// TIA Portal V18 export
FUNCTION "AHUTargetUnitStatesCtrl" : Void   // FC60104, LAD
{ S7_Optimized_Access := 'TRUE' }
VERSION : 0.1
// Operation Modes                                                 Unit State
// 0=Protection                                                         0=Stopped
// 1=Economy                                                           1=Checking-up  
// 2=PreComfort                                                       2=Preheating
// 3=Comfor                                                              3=Starting 
// 4=Auto(Scheduler)                                              4=RecirculatingOperation
//                                                                                 5=Economy Operation                                                                                                                                            6=PreComfort Operation 
//                                                                                 7=Comfort  operation
//                                                                                 8=Stopping
//                                                                                 9=Blocking
// stored: AutoNumber false, IsIECCheckEnabled false, SetENOAutomatically false, UDAEnableTagReadback false
   VAR_INPUT
      iUnitID : Int;
      cTargetOpMode : Byte;
      cActualOpMode : Byte;
      xStartRequest : Bool;
      xBlockRequest : Bool;
   END_VAR
   VAR_OUTPUT
      cTargetUnitState : Byte;
   END_VAR
BEGIN

REGION Network 1 (SCL)
   CASE #cActualOpMode OF
       0:                                                  // OpMode is OFF(Protection)
           IF #xBlockRequest THEN                               // Stop by alarm      
               #cTargetUnitState := 9;
           ELSE 
               #cTargetUnitState := 0;
           END_IF;
       1:                                                  // Economy mode 
           IF #xBlockRequest THEN                               // Stop by alarm      
               #cTargetUnitState := 9;
           ELSIF #xStartRequest THEN                           //Time to start
               #cTargetUnitState := 5;
           ELSE                                                // Stop by no request
               #cTargetUnitState := 0;
           END_IF;
       2:                                                  // PreComfort mode 
           IF #xBlockRequest THEN                               // Stop by alarm      
               #cTargetUnitState := 9;
           ELSIF #xStartRequest THEN                           //Time to start
               #cTargetUnitState := 6;
           ELSE                                                // Stop by no request
               #cTargetUnitState := 0;
           END_IF;
       3:                                                      // Comfort mode 
           IF #xBlockRequest THEN                               // Stop by alarm      
               #cTargetUnitState := 9;
           ELSIF #xStartRequest THEN                           //Time to start
               #cTargetUnitState := 7;
           ELSE                                                // Stop by no request
               #cTargetUnitState := 0;
           END_IF;
       ELSE:
           IF #xBlockRequest THEN                               // Stop by alarm      
               #cTargetUnitState := 9;
           ELSE
               #cTargetUnitState := 0;
           END_IF;
   END_CASE;
END_REGION

REGION Network 2 (SCL)
   IF #cTargetUnitState <> "cTargetUnitStatePrevOne" THEN
       "iTargetUnitStareCounter" := "iTargetUnitStareCounter" + 1;
   END_IF;

   "cTargetUnitStatePrevOne" := #cTargetUnitState;
END_REGION
END_FUNCTION
